FUNCTION_BLOCK FB_SlitPairV3
VAR_INPUT
END_VAR
VAR_OUTPUT
END_VAR
VAR
END_VAR

END_FUNCTION_BLOCK

(* stored: Version 1.1.0.1, ProductVersion 3.1.4024.11
   POU FB_SlitPairV3: Id {b824e8ec-7c24-44c0-9185-5af4f0e9e179}, SpecialFunc None *)
